// TIA Portal V17 export
// export: Created 2022-04-06T07:28:39.6037141Z, ExportSetting WithDefaults, DisplayName Totally Integrated Automation Portal, DisplayVersion V17, DisplayName TIA Portal Openness, DisplayVersion V17, DisplayName TIA Portal Version Control Interface, DisplayVersion V17, DisplayName TIA Portal Test Suite Advanced, DisplayVersion V17, DisplayName SINAMICS Startdrive Advanced, DisplayVersion V17, DisplayName SINAMICS Startdrive G130, G150, S120, S150, SINAMICS MV, S210, DisplayVersion V17, DisplayName SINAMICS Startdrive G110M, G120, G120C, G120D, G120P, G115D, DisplayVersion V17, DisplayName STEP 7 Professional, DisplayVersion V17, DisplayName STEP 7 Safety, DisplayVersion V17, DisplayName WinCC Advanced / Unified PC, DisplayVersion V17
DATA_BLOCK "Main_Safety_RTG1_DB"   // DB1, F_DB
NAME : FUSI
VERSION : 0.1
// stored: AutoNumber true, DBAccessibleFromOPCUA true, DBAccessibleFromWebserver true, InstanceOfName Main_Safety_RTG1, InstanceOfType FB
"Main_Safety_RTG1"
   // VAR
   //    instACK_GL : ACK_GL;
   //    instLDrvSafe_SinaTlg901Control_1 : "LDrvSafe_typeSinaTlg901Control";
   //    instLDrvSafe_SinaTlg901Control : "LDrvSafe_SinaTlg901Control";
   //    instLDrvSafe_SinaTlg901Status : "LDrvSafe_SinaTlg901Status";
   //    instLDrvSafe_SinaSTlg30Control2 : "LDrvSafe_SinaSTlg30Control";
   //    instLDrvSafe_SinaSTlg30Status2 : "LDrvSafe_SinaSTlg30Status";
   //    instSINA_FFB : "SINA_FFB";
   //    instSINA_FFB1 : "SINA_FFB1";
   // END_VAR
BEGIN
END_DATA_BLOCK
